TYPE ST125_Feeder_e : ST110_Feeder_e;
END_TYPE

(* stored: Version 1.1.0.1, ProductVersion 3.1.4024.6
   DUT ST125_Feeder_e: Id {50be5398-8945-4d3a-9abf-e76a9a17b067} *)
